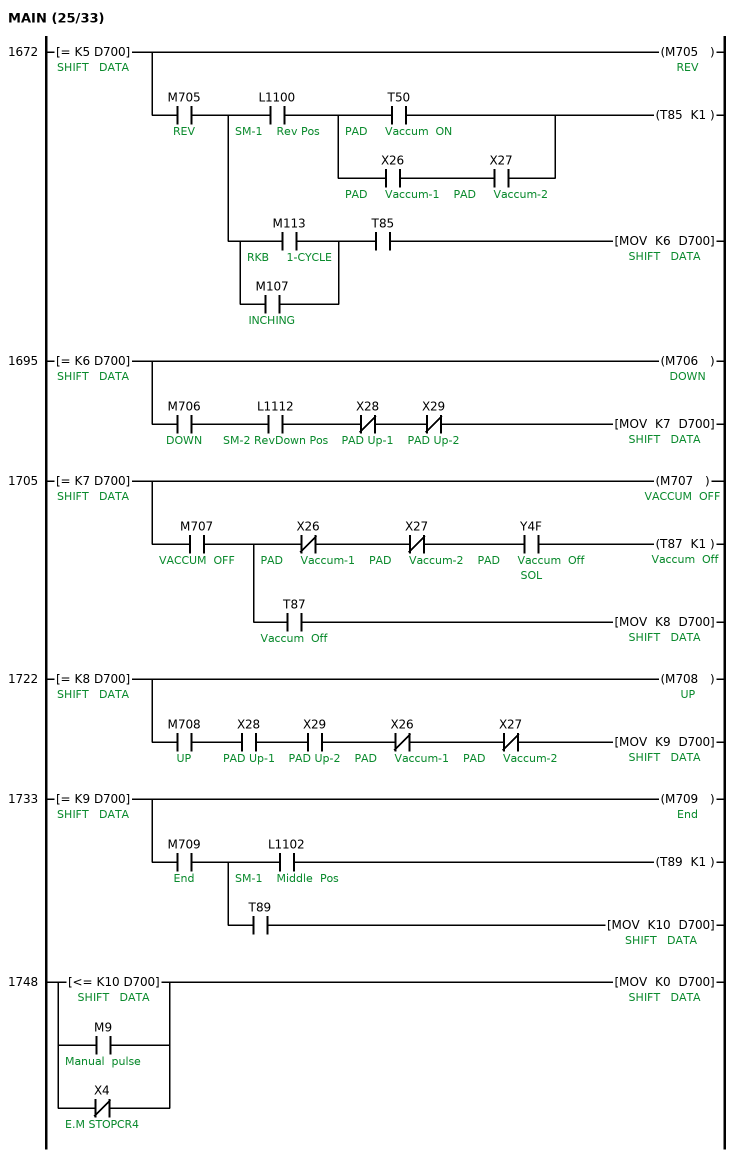
[picture p24: ladder of MAIN, rungs at steps 1672 to 1748]
1672  LD=     K5 D700  ; SHIFT   DATA
      OUT     M705  ; REV
      AND     M705  ; REV
      MPS
      AND     L1100  ; SM-1    Rev Pos
      LD      T50  ; PAD     Vaccum  ON
      LD      X26  ; PAD     Vaccum-1
      AND     X27  ; PAD     Vaccum-2
      ORB
      ANB
      OUT     T85 K1
      MPP
      LD      M113  ; RKB     1-CYCLE
      OR      M107  ; INCHING
      ANB
      AND     T85
      MOV     K6 D700
1695  LD=     K6 D700  ; SHIFT   DATA
      OUT     M706  ; DOWN
      AND     M706  ; DOWN
      AND     L1112  ; SM-2 RevDown Pos
      ANI     X28  ; PAD Up-1
      ANI     X29  ; PAD Up-2
      MOV     K7 D700
1705  LD=     K7 D700  ; SHIFT   DATA
      OUT     M707  ; VACCUM  OFF
      AND     M707  ; VACCUM  OFF
      MPS
      ANI     X26  ; PAD     Vaccum-1
      ANI     X27  ; PAD     Vaccum-2
      AND     Y4F  ; PAD     Vaccum  Off SOL
      OUT     T87 K1  ; Vaccum  Off
      MPP
      AND     T87  ; Vaccum  Off
      MOV     K8 D700
1722  LD=     K8 D700  ; SHIFT   DATA
      OUT     M708  ; UP
      AND     M708  ; UP
      AND     X28  ; PAD Up-1
      AND     X29  ; PAD Up-2
      ANI     X26  ; PAD     Vaccum-1
      ANI     X27  ; PAD     Vaccum-2
      MOV     K9 D700
1733  LD=     K9 D700  ; SHIFT   DATA
      OUT     M709  ; End
      AND     M709  ; End
      MPS
      AND     L1102  ; SM-1    Middle  Pos
      OUT     T89 K1
      MPP
      AND     T89
      MOV     K10 D700
1748  LD<=    K10 D700  ; SHIFT   DATA
      OR      M9  ; Manual  pulse
      ORI     X4  ; E.M STOPCR4
      MOV     K0 D700
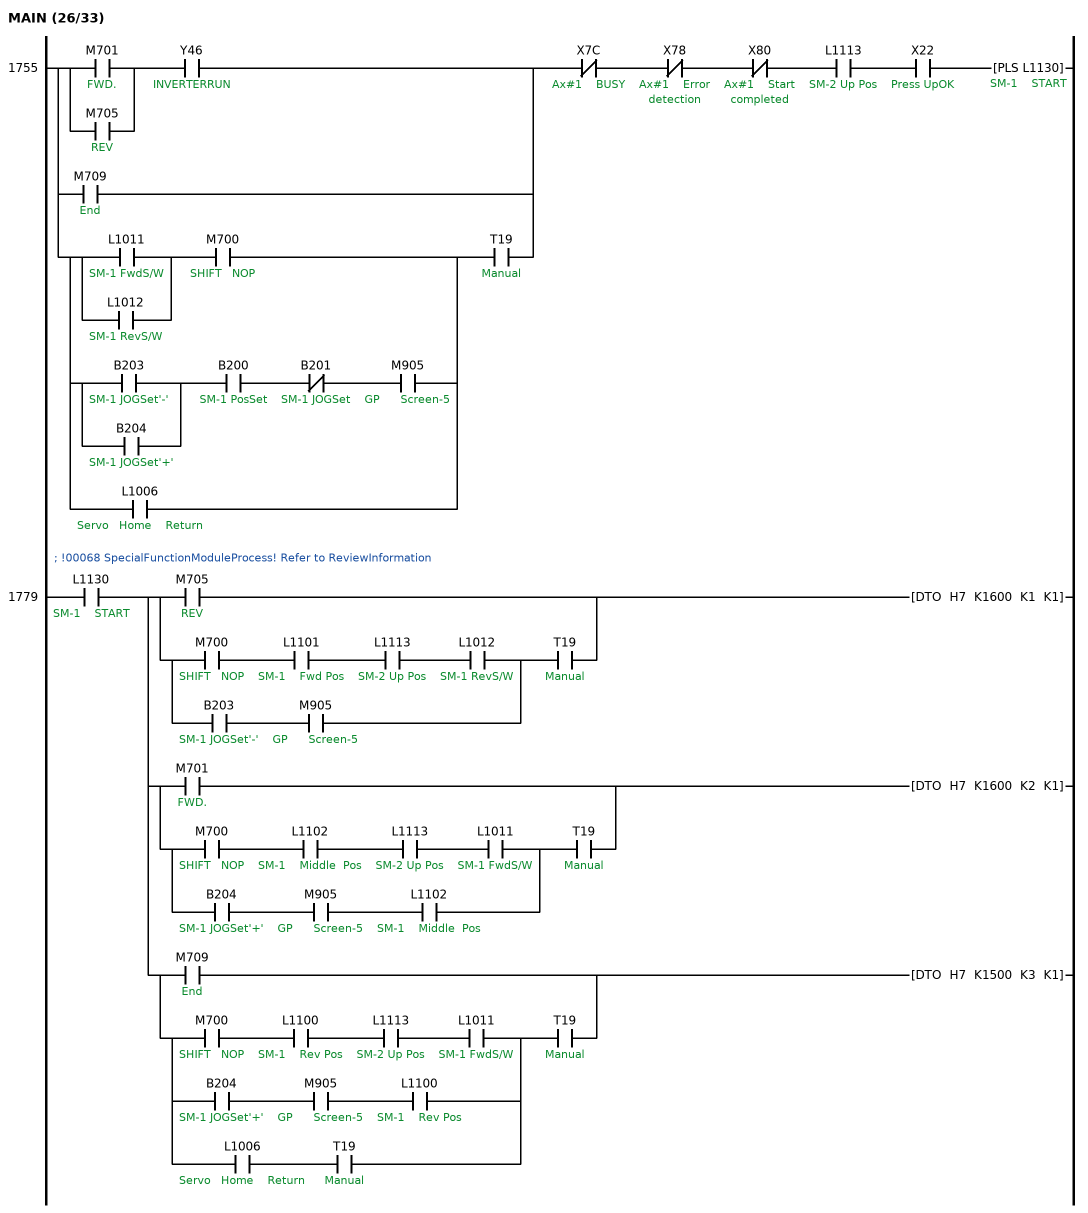
1755  LD      M701  ; FWD.
      OR      M705  ; REV
      AND     Y46  ; INVERTERRUN
      OR      M709  ; End
      LD      L1011  ; SM-1 FwdS/W
      OR      L1012  ; SM-1 RevS/W
      AND     M700  ; SHIFT   NOP
      LD      B203  ; SM-1 JOGSet'-'
      OR      B204  ; SM-1 JOGSet'+'
      AND     B200  ; SM-1 PosSet
      ANI     B201  ; SM-1 JOGSet
      AND     M905  ; GP      Screen-5
      ORB
      OR      L1006  ; Servo   Home    Return
      AND     T19  ; Manual
      ORB
      ANI     X7C  ; Ax#1    BUSY
      ANI     X78  ; Ax#1    Error   detection
      ANI     X80  ; Ax#1    Start   completed
      AND     L1113  ; SM-2 Up Pos
      AND     X22  ; Press UpOK
      PLS     L1130  ; SM-1    START
; !00068 SpecialFunctionModuleProcess! Refer to ReviewInformation
1779  LD      L1130  ; SM-1    START
      MPS
      LD      M705  ; REV
      LD      M700  ; SHIFT   NOP
      AND     L1101  ; SM-1    Fwd Pos
      AND     L1113  ; SM-2 Up Pos
      AND     L1012  ; SM-1 RevS/W
      LD      B203  ; SM-1 JOGSet'-'
      AND     M905  ; GP      Screen-5
      ORB
      AND     T19  ; Manual
      ORB
      ANB
      DTO     H7 K1600 K1 K1
      MRD
      LD      M701  ; FWD.
      LD      M700  ; SHIFT   NOP
      AND     L1102  ; SM-1    Middle  Pos
      AND     L1113  ; SM-2 Up Pos
      AND     L1011  ; SM-1 FwdS/W
      LD      B204  ; SM-1 JOGSet'+'
      AND     M905  ; GP      Screen-5
      AND     L1102  ; SM-1    Middle  Pos
      ORB
      AND     T19  ; Manual
      ORB
      ANB
      DTO     H7 K1600 K2 K1
      MPP
      LD      M709  ; End
      LD      M700  ; SHIFT   NOP
      AND     L1100  ; SM-1    Rev Pos
      AND     L1113  ; SM-2 Up Pos
      AND     L1011  ; SM-1 FwdS/W
      LD      B204  ; SM-1 JOGSet'+'
      AND     M905  ; GP      Screen-5
      AND     L1100  ; SM-1    Rev Pos
      ORB
      LD      L1006  ; Servo   Home    Return
      AND     T19  ; Manual
      ORB
      AND     T19  ; Manual
      ORB
      ANB
      DTO     H7 K1500 K3 K1
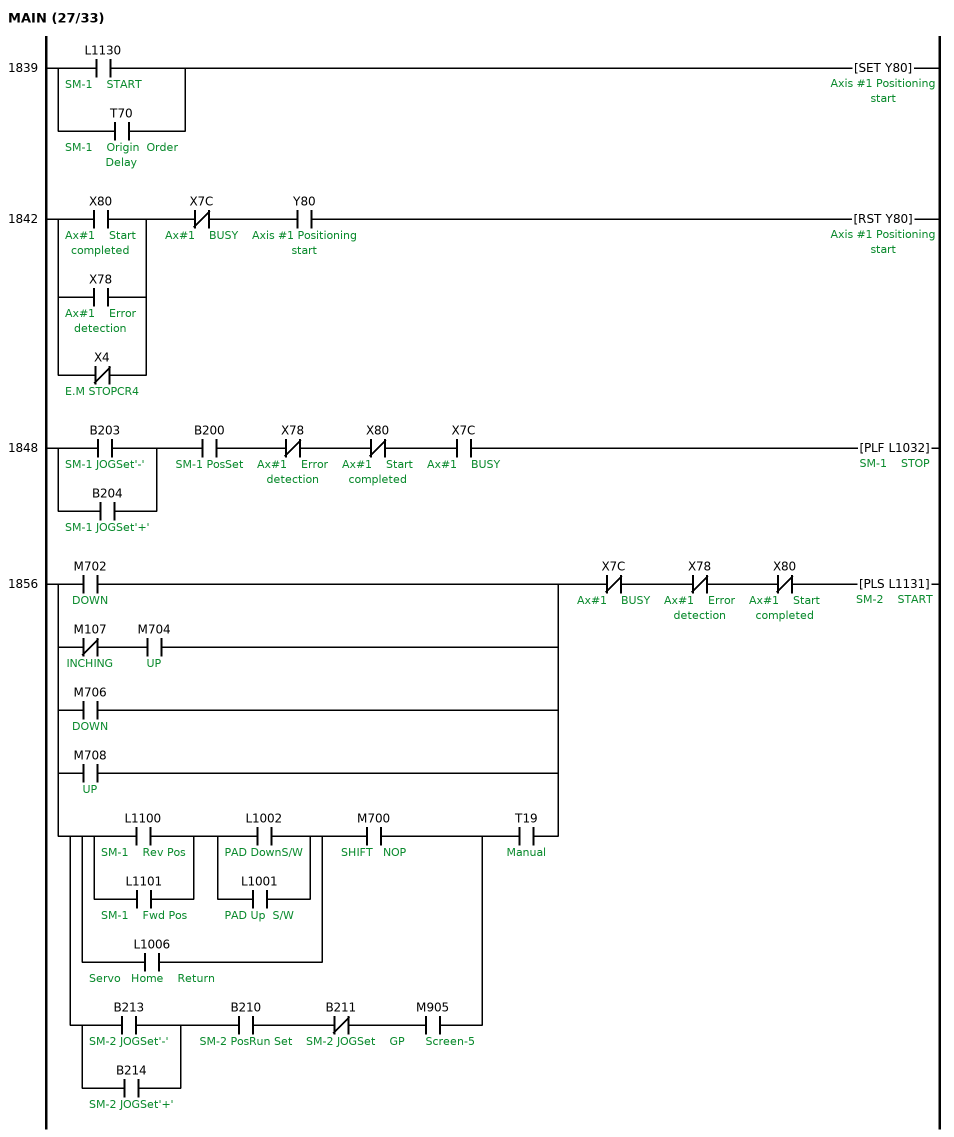
1839  LD      L1130  ; SM-1    START
      OR      T70  ; SM-1    Origin  Order   Delay
      SET     Y80  ; Axis #1 Positioning start
1842  LD      X80  ; Ax#1    Start   completed
      OR      X78  ; Ax#1    Error   detection
      ORI     X4  ; E.M STOPCR4
      ANI     X7C  ; Ax#1    BUSY
      AND     Y80  ; Axis #1 Positioning start
      RST     Y80  ; Axis #1 Positioning start
1848  LD      B203  ; SM-1 JOGSet'-'
      OR      B204  ; SM-1 JOGSet'+'
      AND     B200  ; SM-1 PosSet
      ANI     X78  ; Ax#1    Error   detection
      ANI     X80  ; Ax#1    Start   completed
      AND     X7C  ; Ax#1    BUSY
      PLF     L1032  ; SM-1    STOP
1856  LD      M702  ; DOWN
      LDI     M107  ; INCHING
      AND     M704  ; UP
      ORB
      OR      M706  ; DOWN
      OR      M708  ; UP
      LD      L1100  ; SM-1    Rev Pos
      OR      L1101  ; SM-1    Fwd Pos
      LD      L1002  ; PAD DownS/W
      OR      L1001  ; PAD Up  S/W
      ANB
      OR      L1006  ; Servo   Home    Return
      AND     M700  ; SHIFT   NOP
      LD      B213  ; SM-2 JOGSet'-'
      OR      B214  ; SM-2 JOGSet'+'
      AND     B210  ; SM-2 PosRun Set
      ANI     B211  ; SM-2 JOGSet
      AND     M905  ; GP      Screen-5
      ORB
      AND     T19  ; Manual
      ORB
      ANI     X7C  ; Ax#1    BUSY
      ANI     X78  ; Ax#1    Error   detection
      ANI     X80  ; Ax#1    Start   completed
      PLS     L1131  ; SM-2    START
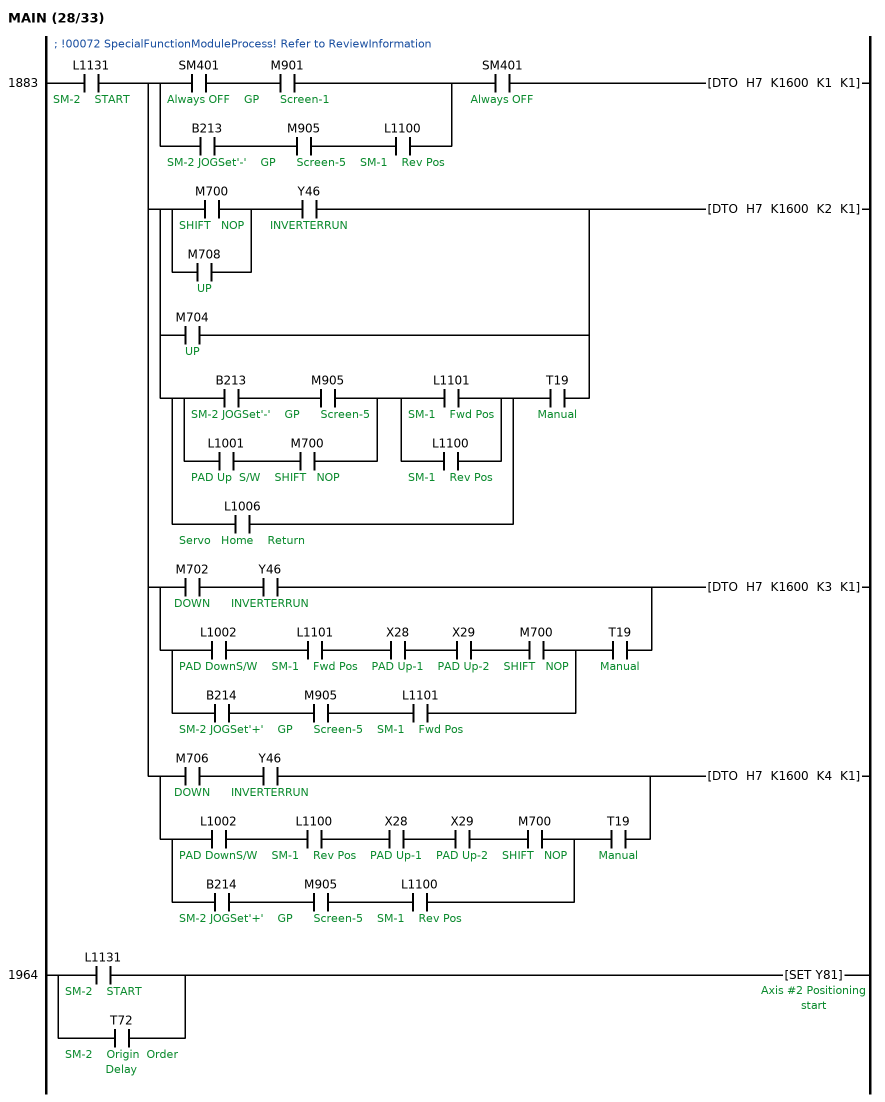
; !00072 SpecialFunctionModuleProcess! Refer to ReviewInformation
1883  LD      L1131  ; SM-2    START
      MPS
      LD      SM401  ; Always OFF
      AND     M901  ; GP      Screen-1
      LD      B213  ; SM-2 JOGSet'-'
      AND     M905  ; GP      Screen-5
      AND     L1100  ; SM-1    Rev Pos
      ORB
      ANB
      AND     SM401  ; Always OFF
      DTO     H7 K1600 K1 K1
      MRD
      LD      M700  ; SHIFT   NOP
      OR      M708  ; UP
      AND     Y46  ; INVERTERRUN
      OR      M704  ; UP
      LD      B213  ; SM-2 JOGSet'-'
      AND     M905  ; GP      Screen-5
      LD      L1001  ; PAD Up  S/W
      AND     M700  ; SHIFT   NOP
      ORB
      LD      L1101  ; SM-1    Fwd Pos
      OR      L1100  ; SM-1    Rev Pos
      ANB
      OR      L1006  ; Servo   Home    Return
      AND     T19  ; Manual
      ORB
      ANB
      DTO     H7 K1600 K2 K1
      MRD
      LD      M702  ; DOWN
      AND     Y46  ; INVERTERRUN
      LD      L1002  ; PAD DownS/W
      AND     L1101  ; SM-1    Fwd Pos
      AND     X28  ; PAD Up-1
      AND     X29  ; PAD Up-2
      AND     M700  ; SHIFT   NOP
      LD      B214  ; SM-2 JOGSet'+'
      AND     M905  ; GP      Screen-5
      AND     L1101  ; SM-1    Fwd Pos
      ORB
      AND     T19  ; Manual
      ORB
      ANB
      DTO     H7 K1600 K3 K1
      MPP
      LD      M706  ; DOWN
      AND     Y46  ; INVERTERRUN
      LD      L1002  ; PAD DownS/W
      AND     L1100  ; SM-1    Rev Pos
      AND     X28  ; PAD Up-1
      AND     X29  ; PAD Up-2
      AND     M700  ; SHIFT   NOP
      LD      B214  ; SM-2 JOGSet'+'
      AND     M905  ; GP      Screen-5
      AND     L1100  ; SM-1    Rev Pos
      ORB
      AND     T19  ; Manual
      ORB
      ANB
      DTO     H7 K1600 K4 K1
1964  LD      L1131  ; SM-2    START
      OR      T72  ; SM-2    Origin  Order   Delay
      SET     Y81  ; Axis #2 Positioning start
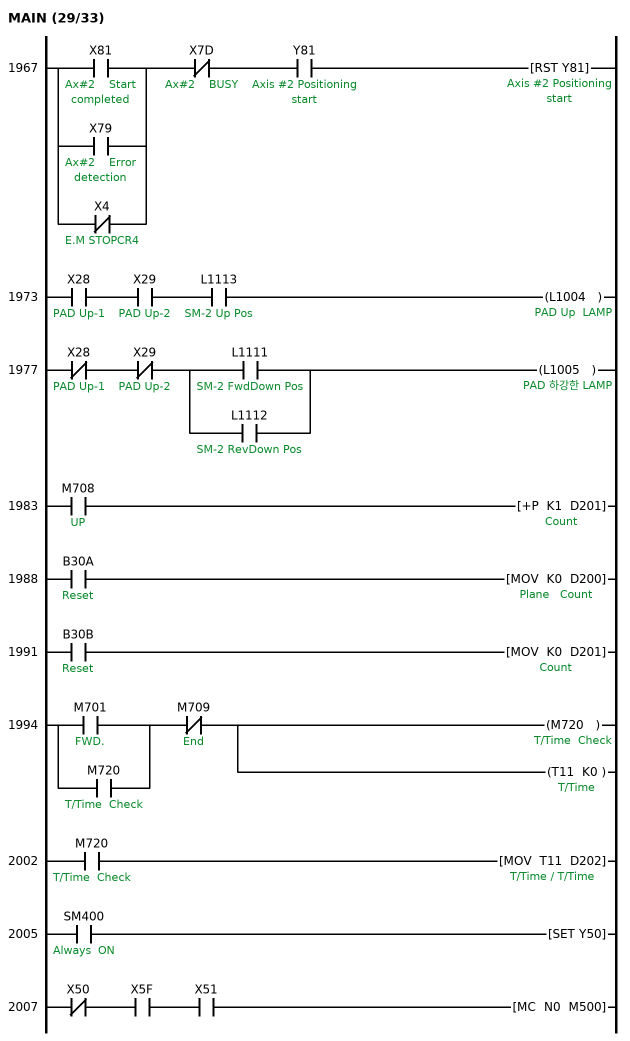
1967  LD      X81  ; Ax#2    Start   completed
      OR      X79  ; Ax#2    Error   detection
      ORI     X4  ; E.M STOPCR4
      ANI     X7D  ; Ax#2    BUSY
      AND     Y81  ; Axis #2 Positioning start
      RST     Y81  ; Axis #2 Positioning start
1973  LD      X28  ; PAD Up-1
      AND     X29  ; PAD Up-2
      AND     L1113  ; SM-2 Up Pos
      OUT     L1004  ; PAD Up  LAMP
1977  LDI     X28  ; PAD Up-1
      ANI     X29  ; PAD Up-2
      LD      L1111  ; SM-2 FwdDown Pos
      OR      L1112  ; SM-2 RevDown Pos
      ANB
      OUT     L1005  ; PAD 하강한 LAMP
1983  LD      M708  ; UP
      +P      K1 D201  ; Count
1988  LD      B30A  ; Reset
      MOV     K0 D200  ; Plane   Count
1991  LD      B30B  ; Reset
      MOV     K0 D201
1994  LD      M701  ; FWD.
      OR      M720  ; T/Time  Check
      ANI     M709  ; End
      OUT     M720  ; T/Time  Check
      OUT     T11 K0  ; T/Time
2002  LD      M720  ; T/Time  Check
      MOV     T11 D202  ; T/Time
2005  LD      SM400  ; Always  ON
      SET     Y50
2007  LDI     X50
      AND     X5F
      AND     X51
      MC      N0 M500
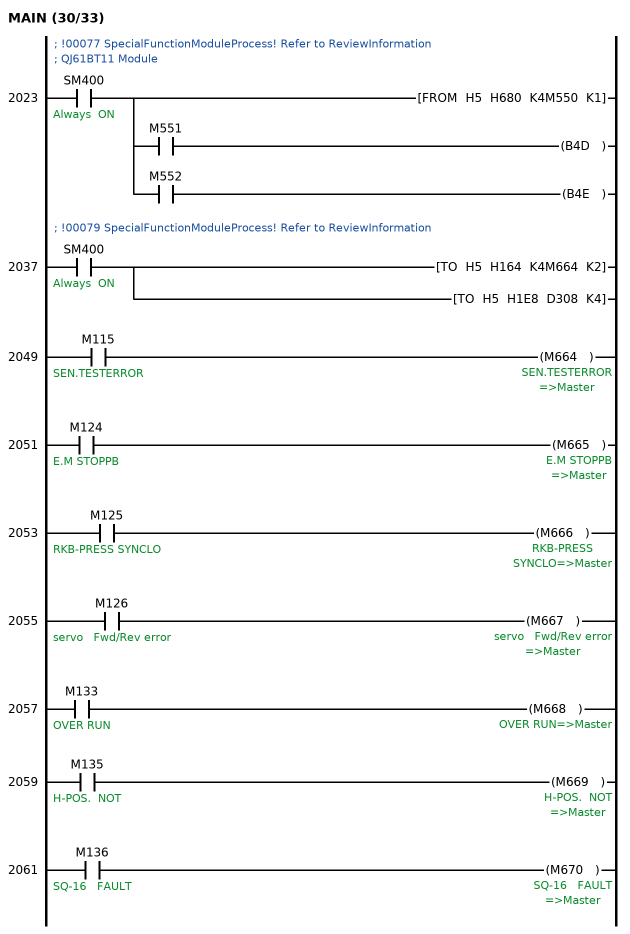
; !00077 SpecialFunctionModuleProcess! Refer to ReviewInformation
; QJ61BT11 Module
2023  LD      SM400  ; Always  ON
      FROM    H5 H680 K4M550 K1
      MPS
      AND     M551
      OUT     B4D
      MPP
      AND     M552
      OUT     B4E
; !00079 SpecialFunctionModuleProcess! Refer to ReviewInformation
2037  LD      SM400  ; Always  ON
      TO      H5 H164 K4M664 K2  ; SEN.TESTERROR   =>Master
      TO      H5 H1E8 D308 K4
2049  LD      M115  ; SEN.TESTERROR
      OUT     M664  ; SEN.TESTERROR   =>Master
2051  LD      M124  ; E.M STOPPB
      OUT     M665  ; E.M STOPPB      =>Master
2053  LD      M125  ; RKB-PRESS SYNCLO
      OUT     M666  ; RKB-PRESS SYNCLO=>Master
2055  LD      M126  ; servo   Fwd/Rev error
      OUT     M667  ; servo   Fwd/Rev error   =>Master
2057  LD      M133  ; OVER RUN
      OUT     M668  ; OVER RUN=>Master
2059  LD      M135  ; H-POS.  NOT
      OUT     M669  ; H-POS.  NOT     =>Master
2061  LD      M136  ; SQ-16   FAULT
      OUT     M670  ; SQ-16   FAULT   =>Master
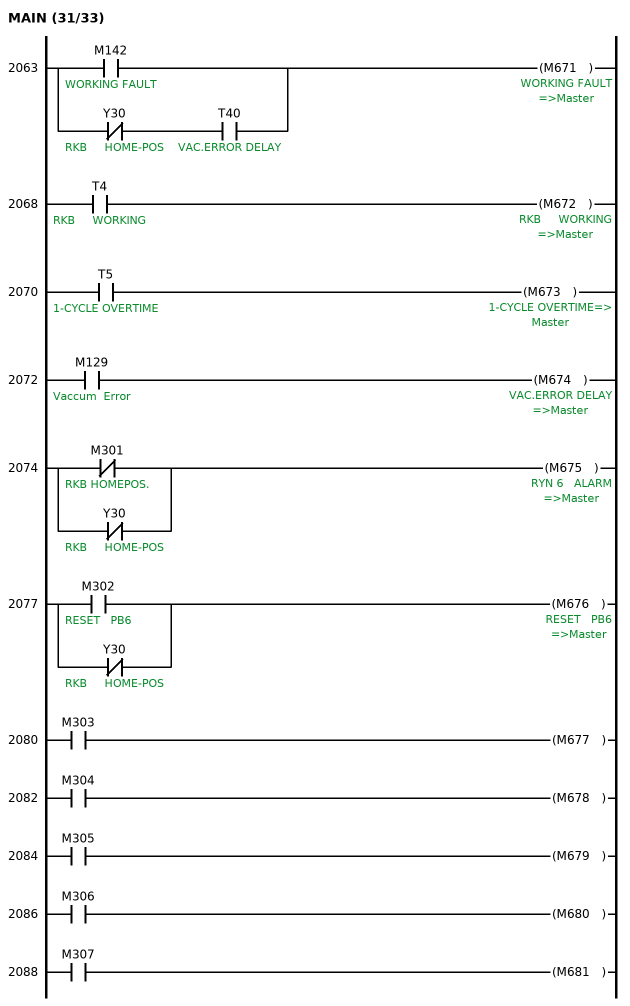
2063  LD      M142  ; WORKING FAULT
      LDI     Y30  ; RKB     HOME-POS
      AND     T40  ; VAC.ERROR DELAY
      ORB
      OUT     M671  ; WORKING FAULT   =>Master
2068  LD      T4  ; RKB     WORKING
      OUT     M672  ; RKB     WORKING =>Master
2070  LD      T5  ; 1-CYCLE OVERTIME
      OUT     M673  ; 1-CYCLE OVERTIME=>Master
2072  LD      M129  ; Vaccum  Error
      OUT     M674  ; VAC.ERROR DELAY =>Master
2074  LDI     M301  ; RKB HOMEPOS.
      ORI     Y30  ; RKB     HOME-POS
      OUT     M675  ; RYN 6   ALARM   =>Master
2077  LD      M302  ; RESET   PB6
      ORI     Y30  ; RKB     HOME-POS
      OUT     M676  ; RESET   PB6     =>Master
2080  LD      M303
      OUT     M677
2082  LD      M304
      OUT     M678
2084  LD      M305
      OUT     M679
2086  LD      M306
      OUT     M680
2088  LD      M307
      OUT     M681
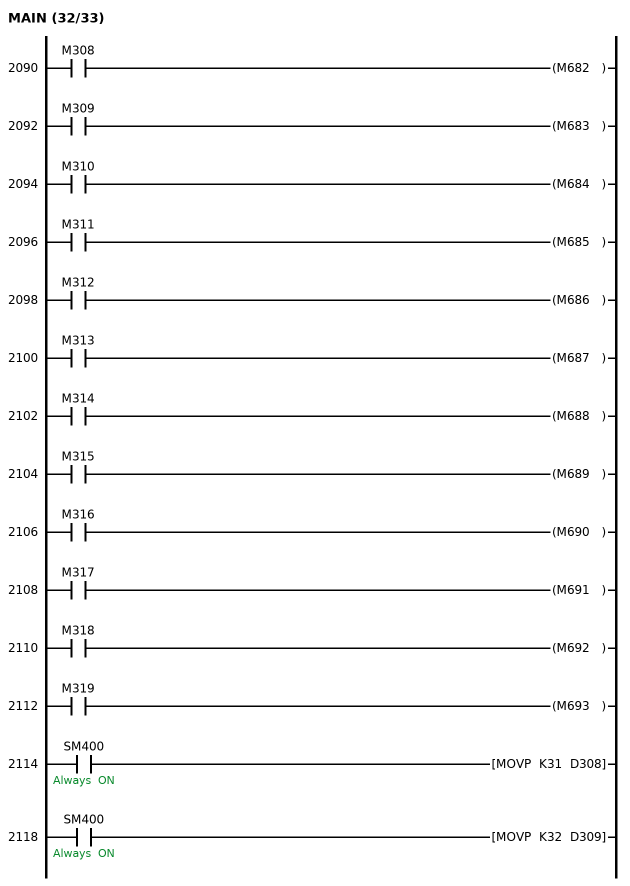
2090  LD      M308
      OUT     M682
2092  LD      M309
      OUT     M683
2094  LD      M310
      OUT     M684
2096  LD      M311
      OUT     M685
2098  LD      M312
      OUT     M686
2100  LD      M313
      OUT     M687
2102  LD      M314
      OUT     M688
2104  LD      M315
      OUT     M689
2106  LD      M316
      OUT     M690
2108  LD      M317
      OUT     M691
2110  LD      M318
      OUT     M692
2112  LD      M319
      OUT     M693
2114  LD      SM400  ; Always  ON
      MOVP    K31 D308
2118  LD      SM400  ; Always  ON
      MOVP    K32 D309
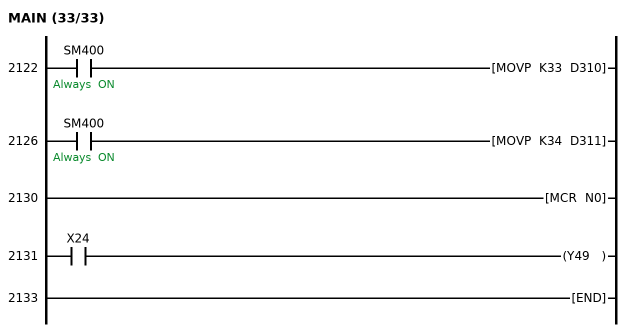
2122  LD      SM400  ; Always  ON
      MOVP    K33 D310
2126  LD      SM400  ; Always  ON
      MOVP    K34 D311
2130  MCR     N0
2131  LD      X24
      OUT     Y49
2133  END
END_PROGRAM

// device comments not shown above
M114  ; VAC.    ERROR
M150  ; LOW AIR PRESSURE
M155  ; QUICK   RELEASE
X10  ; RKB     HOME-POS
X12  ; 1-CYCLE STOP
X13  ; VACUUM  FOR WORK
X14  ; SEN.TESTSPHERE
X16  ; INCH.   FWD END
X17  ; INCH.   REV END
X1B  ; SQ-12   RUN
X1C  ; QUICK RELEASE SE
X71  ; Synchronization flag
X74  ; Ax#1 M code ON
X75  ; Ax#2 M code ON
X76  ; Ax#3 M code ON
X77  ; Ax#4 M code ON
X7A  ; Ax#3 Error detection
X7B  ; Ax#4 Error detection
X7E  ; Ax#3 BUSY
X7F  ; Ax#4 BUSY
X82  ; Ax#3 Start completed
X83  ; Ax#4 Start completed
X84  ; Ax#1 Positioning completed
X85  ; Ax#2 Positioning completed
X86  ; Ax#3 Positioning completed
X87  ; Ax#4 Positioning completed
Y36  ; MOTOR   BRAKE
Y76  ; Ax#3 Axis stop
Y77  ; Ax#4 Axis stop
Y7C  ; Ax#3 Forward rotation JOG start
Y7D  ; Ax#3 Reverse rotation JOG start
Y7E  ; Ax#4 Forward rotation JOG start
Y7F  ; Ax#4 Reverse rotation JOG start
Y82  ; Axis #3 Positioning start
Y83  ; Axis #4 Positioning start
Y84  ; Ax#1 Execution prohibition flag
Y85  ; Ax#2 Execution prohibition flag
Y86  ; Ax#3 Execution prohibition flag
Y87  ; Ax#4 Execution prohibition flag
